(* IEC 61131-3 sources: crb-codesys/retrieval/output/codesys_repo/PID_controller/Progs, 3 files *)

(* ---- Test_PID.st ---- *)
PROGRAM Test_PID
VAR
	PID_0: PID_controller;
	RedBull: Tank;
	Process_out: REAL := 100;
	SetPoint: REAL := 250;
END_VAR

VAR CONSTANT
END_VAR

PID_0(
    SP := SetPoint,                // 设定值：目标液位250
    PV := RedBull.Level,              // 过程值：储罐当前液位（反馈）
    Kc := 2,                  // 比例增益2.0
    Ti := 15,                  // 积分时间15.0
    Td := 1,                  // 微分时间1.0
    SampleTime := T#100ms,  // 采样时间100ms
    LowerLimit := 0,  // 输出下限0
    UpperLimit := 150,  // 输出上限150
    CO => ,                  // PID输出：控制储罐的输入流量
    CO_P => ,                      // 比例部分输出（未使用可留空）
    CO_I => ,                      // 积分部分输出（未使用可留空）
    CO_D =>                        // 微分部分输出（未使用可留空）
);

// 2. 调用储罐功能块
RedBull(
    Process_In := PID_0.CO,          // 输入流量：PID的输出CO
    Process_Out := Process_out,    // 输出流量：100（外部定义）
    Sample_time := T#250ms,// 采样时间250ms
    Lower_limit := 0,// 液位下限0
    Upper_limit := 500,// 液位上限500
    Level =>             // 输出当前液位：反馈给PID的PV
);

(* ---- Test_PID_Heat2.st ---- *)
PROGRAM Test_PID_Heat2
VAR
	PID_controller_0: PID_controller;
	HeatExchanger2_0: HeatExchanger2;
	SP: REAL := 300;
	Temp_out: REAL := 270;
END_VAR

PID_controller_0(
    SP := SP,                // 设定值：目标液位250
    PV := HeatExchanger2_0.Temp,              // 过程值：储罐当前液位（反馈）
    Kc := 50,                  // 比例增益2.0
    Ti := 5,                  // 积分时间15.0
    Td := 0,                  // 微分时间1.0
    SampleTime := T#250ms,  // 采样时间100ms
    LowerLimit := 0,  // 输出下限0
    UpperLimit := 6000,  // 输出上限150
    CO => ,                  // PID输出：控制储罐的输入流量
    CO_P => ,                      // 比例部分输出（未使用可留空）
    CO_I => ,                      // 积分部分输出（未使用可留空）
    CO_D =>                        // 微分部分输出（未使用可留空）
);

// 2. 调用储罐功能块
HeatExchanger2_0(
    Heat_In := PID_controller_0.CO,
    U := 100,
    TC := 2500,
    Temp_In := 270,
    Temp_Out := Temp_Out;
    Sample_time := T#100ms,
    Temp =>
);

(* ---- Test_PID_Heatx.st ---- *)
PROGRAM Test_PID_Heatx
VAR
	PID_0: PID_controller;
	Process_out: REAL := 100;
	SetPoint: REAL := 20;
	A_room_with_a_view: HeatExchanger;
END_VAR

VAR CONSTANT
END_VAR

PID_0(
    SP := SetPoint,
    PV := A_room_with_a_view.PV,
    Kc := 5.0,
    Ti := 10.0,
    Td := 1.0,
    SampleTime := T#2000ms,
    LowerLimit := 0,
    UpperLimit := 150,
    CO => ,  // 若不需要单独使用 CO 等输出，可留空，或根据需求定义变量接收
    CO_P => ,
    CO_I => ,
    CO_D =>
);

// 调用 HeatExchanger 功能块
A_room_with_a_view(
    Kp := 2.0,
    Tp := 20,
    CO := PID_0.CO,
    Dead_t := 9.8,
    C := 2.048,
    Sample_time := T#100ms,
    PV =>
);
